FUNCTION_BLOCK MotorS (* CAT Function Block Type *)
  (* Standard: 61499-2 *)
  (* Version 0.0, 6/2/2026, Schneider Electric, template *)
  PACKAGE SE.Nereda;
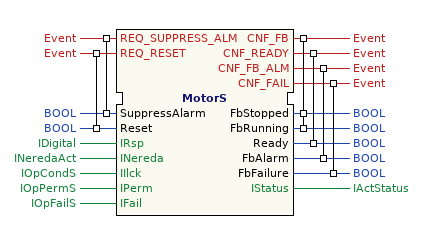
  EVENT_INPUT
    REQ_SUPPRESS_ALM WITH SuppressAlarm; (* Request to update the alarm suppress status *)
    REQ_RESET WITH Reset; (* Request to reset the device *)
  END_EVENT
  EVENT_OUTPUT
    CNF_FB WITH FbStopped, FbRunning; (* Execution of confirmed state *)
    CNF_READY WITH Ready; (* Execution of Ready status *)
    CNF_FB_ALM WITH FbAlarm; (* Execution of confirmation  Fb alarm *)
    CNF_FAIL WITH FbFailure; (* Execution of confirmation  failure *)
  END_EVENT
  VAR_INPUT
    SuppressAlarm : BOOL; (* 1 = Suppress alarm in HMI *)
    Reset : BOOL; (* 1 = Reset device failure *)
  END_VAR
  VAR_OUTPUT
    FbStopped : BOOL; (* 1 = Stopped *)
    FbRunning : BOOL; (* 1 = Running *)
    Ready : BOOL; (* 1 = Device is ready to run *)
    FbAlarm : BOOL; (* 1 = Feedback failure alarm is active *)
    FbFailure : BOOL; (* 1 = Fail active *)
  END_VAR
  SOCKETS
    IRsp : IDigital;
    INereda : INeredaAct;
  END_SOCKETS
  SOCKETS
    IIlck : IOpCondS; (* Condition summary chain input from upstream blocks *)
    IPerm : IOpPermS; (* Permission condition summary chain input from permCondItem blocks *)
    IFail : IOpFailS; (* Fail condition summary chain input from failCondItem blocks *)
  END_SOCKETS
  PLUGS
    IStatus : IActStatus;
  END_PLUGS
  (* 01 - FUNCTIONNAL INPUT INTERFACE *)
  (* 00 - INITIALIZATION *)
  (* 05 - LOGIC *)
  (* 06 - HMI INTERFACE *)
  (* 04 - CHILDREN *)
  (* 03 - FIELD INTERFACE *)
  (* 02 - FUNCTIONNAL OUTPUT INTERFACE *)
  (* 07- Input Hardware Interface *)
  (* 08- Output Hardware Interface *)
  (* 09- Local Panel *)
  (* Maintenance *)
  (* Fb Stop *)
  (* Interlock *)
  (* Mode *)
  (* Permissive *)
  (* 4A - TYPICALS *)
  (* Craeted By Nouriddin OUECHEN *)
  (* Failure *)
  (* Reset *)
  (* Cmd *)
  (* Comment When `SafetySwitchOff = TRUE`, it means that the safety switch is **OFF**. *)
  FBS
    Base : MotorBase;
    IThis : MotorS_HMI(QI := TRUE);
    INIT : plcStart(Prio := 35, Delay := T#0ms);
    fbRun : dISignal(Name := '$${PATH}DIn'); {SET_ATTRIBUTE(Configuration.Component.HideUnusedPorts, )}
    extControlled : dISignal(Name := '$${PATH}DIn'); {SET_ATTRIBUTE(Configuration.Component.HideUnusedPorts, )}
    cmd : dOSignal(Name := '$${PATH}DOut'); {SET_ATTRIBUTE(Configuration.Component.HideUnusedPorts, )}
    LocalPanel : FieldSignals;
    maintenance : DevMnt(StateSel := Motor); {SET_ATTRIBUTE(Configuration.Component.HideUnusedPorts, )}
    FbStop : NOT_42C76073DCEB1A7A; {SET_ATTRIBUTE(Configuration.GenericFBType.InterfaceParams, Runtime.Standard#CNT:=1;OUT${CNT$}:BOOL)}
    interlock : IlckCondSum; {SET_ATTRIBUTE(Configuration.Component.HideUnusedPorts, )}
    failure : FailCondSum; {SET_ATTRIBUTE(Configuration.Component.HideUnusedPorts, )}
    DriveFailure : failCondItem(CondCause := Active1); {SET_ATTRIBUTE(Configuration.Component.HideUnusedPorts, )}
    AtvFailure : SELECT_81F91C08E00C8B28(IN1 := FALSE); {SET_ATTRIBUTE(Configuration.GenericFBType.InterfaceParams, Runtime.Standard#CNT:=2;SELECT:BOOL;IN${CNT$}:BOOL)}
    ElectricCircuitFailure : failCondItem(CondCause := Active1); {SET_ATTRIBUTE(Configuration.Component.HideUnusedPorts, )}
    FrequencyInverterFailure : failCondItem(CondCause := Active1); {SET_ATTRIBUTE(Configuration.Component.HideUnusedPorts, )}
    PowerFailure : failCondItem(CondCause := Active1); {SET_ATTRIBUTE(Configuration.Component.HideUnusedPorts, )}
    CurrOwner : CurrOwnerDecode;
    State : ActState(pin_DD241BABAE81E6FD := Motor);
    NoPowerFb : NOT_42C76073DCEB1A7A; {SET_ATTRIBUTE(Configuration.GenericFBType.InterfaceParams, Runtime.Standard#CNT:=1;OUT${CNT$}:BOOL)}
    permissive : PermCondSum; {SET_ATTRIBUTE(Configuration.Component.HideUnusedPorts, )}
    ResetCmd : OR_550FE6D62F509EB3; {SET_ATTRIBUTE(Configuration.GenericFBType.InterfaceParams, Runtime.Standard#CNT:=3;OUT:BOOL)}
    Sp : DS_SELECTX_6147A5438F26867; {SET_ATTRIBUTE(Configuration.GenericFBType.InterfaceParams, Runtime.Standard#CNTX:=2;CNTY:=1;DI${CNTX,_,CNTY$}:INT)}
    TRIP : failCondItem(CondCause := Active1); {SET_ATTRIBUTE(Configuration.Component.HideUnusedPorts, )}
    MoistureDetectionPumpMS : failCondItem(CondCause := Active1); {SET_ATTRIBUTE(Configuration.Component.HideUnusedPorts, )}
    INT2BOOL_Cmd : INT2BOOL;
    SafetySwitchOff : ilckCondItem(CondCause := Active1);
    SafetySwitch : NOT_42C76073DCEB1A7A; {SET_ATTRIBUTE(Configuration.GenericFBType.InterfaceParams, Runtime.Standard#CNT:=1;OUT${CNT$}:BOOL)}
    AllFailures : OR_1147623A96AA66A8; {SET_ATTRIBUTE(Configuration.GenericFBType.InterfaceParams, Runtime.Standard#CNT:=7;OUT:BOOL)}
  END_FBS
  EVENT_CONNECTIONS
    extControlled.CNF TO Base.REQ_EXT_CTL;
    fbRun.CNF TO FbStop.REQ;
    FbStop.CNF TO Base.REQ_FB;
    IRsp.REQ TO Sp.REQ1;
    interlock.COND_IND TO Base.REQ_ILCK;
    failure.COND_IND TO Base.REQ_FAIL;
    REQ_SUPPRESS_ALM TO Base.REQ_SUPPRESS_ALM;
    Base.CNF_FB_STS TO CNF_FB;
    Base.CNF_FB_ALM TO CNF_FB_ALM;
    Base.CNF_OUT TO maintenance.REQ;
    Base.CNF_FB_ALM TO maintenance.REQ_ALM;
    Base.CNF_MODE TO maintenance.REQ;
    REQ_SUPPRESS_ALM TO maintenance.REQ_SUPPRESS_ALM;
    NoPowerFb.CNF TO DriveFailure.REQ;
    NoPowerFb.CNF TO ElectricCircuitFailure.REQ;
    NoPowerFb.CNF TO FrequencyInverterFailure.REQ;
    NoPowerFb.CNF TO PowerFailure.REQ;
    permissive.PERM_IND TO Base.REQ_PERM;
    AtvFailure.CNF TO NoPowerFb.REQ;
    Sp.IND TO Base.REQ_SP;
    REQ_RESET TO ResetCmd.REQ;
    ResetCmd.CNF TO Base.REQ_RESET;
    NoPowerFb.CNF TO TRIP.REQ;
    NoPowerFb.CNF TO MoistureDetectionPumpMS.REQ;
    LocalPanel.08EBB16DA2AE2E53 TO AtvFailure.REQ;
    LocalPanel.08EBB16DA2AE2E53 TO AllFailures.REQ;
    INereda.0F1CDF9A9B4A227A TO Sp.REQ2;
    Base.CNF_FB_STS TO INereda.9CD053F8408797ED;
    INereda.37BBC1F841739733 TO ResetCmd.REQ;
    State.3E2F994B40CA5D8A TO INereda.CC753684FA882790;
    Base.CNF_FB_ALM TO INereda.C79FD2A34D0395C5;
    Base.CNF_FAIL TO AllFailures.REQ;
    maintenance.CNF_OPD TO INereda.2DA8AEC15204E92D;
    Base.CNF_SP TO AllFailures.REQ;
    Base.CNF_FB_STS TO AllFailures.REQ;
    Base.CNF_READY TO AllFailures.REQ;
    Base.CNF_OWNER TO AllFailures.REQ;
    Base.CNF_MODE TO AllFailures.REQ;
    interlock.COND_IND TO AllFailures.REQ;
    CurrOwner.7B1DE71047870DF3 TO State.503DFB34A9D9F842;
    State.B9B326A02DDC85D5 TO INIT.ACK_FIRST;
    Base.CNF_OUT TO INT2BOOL_Cmd.DD5870AA881150BB;
    INT2BOOL_Cmd.6FC99A5BD1C38561 TO cmd.REQ;
    Base.CNF_FB_STS TO IStatus.14377629A1F197A9;
    State.3E2F994B40CA5D8A TO IStatus.14377629A1F197A9;
    State.3E2F994B40CA5D8A TO CNF_READY;
    Base.CNF_OWNER TO Base.REQ_SP;
    SafetySwitch.CNF TO SafetySwitchOff.REQ;
    LocalPanel.08EBB16DA2AE2E53 TO SafetySwitch.REQ;
    INIT.FIRST_INIT TO IThis.5D65C7F23F6CCFDB;
    INIT.REDO_INIT TO IThis.5D65C7F23F6CCFDB;
    State.B9B326A02DDC85D5 TO IThis.D29F1FADF6E57358;
    LocalPanel.08EBB16DA2AE2E53 TO IThis.438D25703EEFF814;
    Base.CNF_NEED_RESET TO IThis.56CAC1A52910316B;
    State.7E9F7DF9BBDC513D TO IThis.24BAED5957B7CC26;
    IThis.141F2765F0199247 TO State.747A80A26976E9BA;
    IThis.EDABC861E1C71398 TO AtvFailure.REQ;
    IThis.A591CDF920E284FE TO ResetCmd.REQ;
    State.7E9F7DF9BBDC513D TO CNF_FAIL;
    State.7E9F7DF9BBDC513D TO INereda.476AAA40EB7AA926;
    Base.CNF_FB_ALM TO AllFailures.REQ;
    AllFailures.CNF TO CurrOwner.3D8B91432EBB5812;
    NoPowerFb.CNF TO AllFailures.REQ;
    Base.CNF_NEED_RESET TO AllFailures.REQ;
  END_CONNECTIONS
  DATA_CONNECTIONS
    extControlled.Out TO Base.ExternalControlled;
    fbRun.Out TO Base.FbRun;
    FbStop.OUT1 TO Base.FbStop;
    fbRun.Out TO FbStop.IN1;
    IRsp.Value TO Sp.DI1_1;
    interlock.CondPos TO Base.IlckPos;
    interlock.CondType TO Base.IlckType;
    interlock.State TO Base.IlckCond;
    failure.State TO Base.Fail;
    SuppressAlarm TO Base.SuppressAlarm;
    Base.FbStopped TO FbStopped;
    Base.FbRunning TO FbRunning;
    Base.FbAlarm TO FbAlarm;
    Base.Out TO maintenance.Pv;
    Base.FbAlarm TO maintenance.DeviceAlarm;
    Base.Simulation TO maintenance.Sim;
    SuppressAlarm TO maintenance.SuppressAlarm;
    AtvFailure.OUT TO DriveFailure.CondSignal;
    NoPowerFb.OUT1 TO PowerFailure.CondSignal;
    permissive.PermPassive TO Base.PermStop;
    permissive.PermActive1 TO Base.PermRun;
    Sp.OUT1 TO Base.Sp;
    Reset TO ResetCmd.IN1;
    ResetCmd.OUT TO Base.Reset;
    LocalPanel.9DA3D6735086B77A TO ElectricCircuitFailure.CondSignal;
    LocalPanel.B021B183D08305E2 TO FrequencyInverterFailure.CondSignal;
    LocalPanel.DA445F1C2864A153 TO State.C70237F918BB93F6;
    LocalPanel.B46B24B64003C584 TO NoPowerFb.IN1;
    LocalPanel.B46B24B64003C584 TO State.655DE7D6E2CF8FB8;
    LocalPanel.61B515FEF739774D TO AtvFailure.IN2;
    LocalPanel.4379EE93CED9D91D TO TRIP.CondSignal;
    LocalPanel.5EFEAD483C25BA7B TO MoistureDetectionPumpMS.CondSignal;
    Base.FbStopped TO INereda.D83B5BDEFA4D797C;
    Base.FbRunning TO INereda.B762734C094A7162;
    State.4E509FA35DBACB85 TO INereda.8A8A07EFCDA1443C;
    Base.FbAlarm TO INereda.BDD69968F2D82EAF;
    Base.FailStatus TO AllFailures.IN1;
    maintenance.TotalOperationDuration TO INereda.C7F638DBF6B860D2;
    maintenance.CurrentOperationDuration TO INereda.9224E22E0E82A2D7;
    maintenance.OperationCount TO INereda.10624535249F94F3;
    INereda.710D7FC54EE3F35A TO Sp.DI2_1;
    INereda.EA28053F07575F36 TO ResetCmd.IN3;
    Base.CurrentOwner TO CurrOwner.B2DAC483AB345195;
    CurrOwner.CEBE936F1EA616DB TO State.E90E39DE4A80ABDE;
    CurrOwner.1FF13EB8D921FC26 TO State.3885B231A80F7FFF;
    Base.CurrentSp TO State.52C3EF6D9E750127;
    Base.FbStatus TO State.8E076A9FED13120E;
    Base.Ready TO State.1C9201C719ABF50B;
    Base.Simulation TO State.7A0BDA68B634A263;
    Base.FbOverride TO State.DD66F5DCF7F6FB1D;
    interlock.State TO State.9A204E382C1350DC;
    Base.Out TO INT2BOOL_Cmd.4573FC8F228EB71D;
    INT2BOOL_Cmd.A6DEF5F9C27C1848 TO cmd.Signal;
    Base.FbStopped TO IStatus.227987A2F0C6A825;
    Base.FbRunning TO IStatus.D41A46B14EF7208D;
    State.4E509FA35DBACB85 TO IStatus.9E0B44559326BEAF;
    State.4E509FA35DBACB85 TO Ready;
    SafetySwitch.OUT1 TO SafetySwitchOff.CondSignal;
    LocalPanel.9F4FA80000721942 TO SafetySwitch.IN1;
    LocalPanel.9DA3D6735086B77A TO IThis.0AE962625433D46C;
    LocalPanel.61B515FEF739774D TO IThis.05CEFE840775FD43;
    Base.NeedReset TO IThis.40C9F9C762B4EBFC;
    State.8CCAFBE354ECA569 TO IThis.72E5F23DEBA1B1A4;
    IThis.E887C120F3A4AF42 TO AtvFailure.SELECT;
    IThis.E6FBA099621F55FB TO ResetCmd.IN2;
    State.8CCAFBE354ECA569 TO FbFailure;
    State.8CCAFBE354ECA569 TO INereda.6EEAF63EEE6021B6;
    Base.FbAlarm TO State.F37ACDE435F84908;
    AllFailures.OUT TO State.94E3C396E1CCD1C0;
    AtvFailure.OUT TO AllFailures.IN2;
    NoPowerFb.OUT1 TO AllFailures.IN5;
    LocalPanel.9DA3D6735086B77A TO AllFailures.IN3;
    LocalPanel.B021B183D08305E2 TO AllFailures.IN4;
    LocalPanel.4379EE93CED9D91D TO AllFailures.IN6;
    LocalPanel.5EFEAD483C25BA7B TO AllFailures.IN7;
    Base.NeedReset TO State.3ED730632EF45559;
  END_CONNECTIONS
  ADAPTER_CONNECTIONS
    IIlck TO SafetySwitchOff.ICondChainIn;
    IFail TO DriveFailure.ICondChainIn;
    DriveFailure.ICondChainOut TO ElectricCircuitFailure.ICondChainIn;
    ElectricCircuitFailure.ICondChainOut TO FrequencyInverterFailure.ICondChainIn;
    FrequencyInverterFailure.ICondChainOut TO PowerFailure.ICondChainIn;
    MoistureDetectionPumpMS.ICondChainOut TO failure.IOpCondIn;
    IPerm TO permissive.IOpPermIn;
    PowerFailure.ICondChainOut TO TRIP.ICondChainIn;
    TRIP.ICondChainOut TO MoistureDetectionPumpMS.ICondChainIn;
    SafetySwitchOff.ICondChainOut TO interlock.IOpCondIn;
  END_CONNECTIONS
END_FUNCTION_BLOCK
